{attribute addProperty BoxType "AX8620-0000-0027"}
{attribute addProperty Id "PSM_StatuswordAT %I*PSM_Statusword_C154CB391620WcStateAT %I*WcState_F855686C1620InfoDataAT %I*InfoData_0BDED7BF144180"}
{attribute addProperty CRC "1422836300"}
{attribute addProperty SizeInBites "176"}
{attribute addProperty SizeInBytes "22"}
TYPE AX8620_5E25E4A1 :
STRUCT
	{attribute addProperty Name "PSM_Statusword"}
	PSM_Statusword : PSM_Statusword_C154CB39;
	{attribute addProperty Name "WcState"}
	WcState : WcState_F855686C;
	{attribute addProperty Name "InfoData"}
	InfoData : InfoData_0BDED7BF;
END_STRUCT
END_TYPE

(* stored: Version 1.2.0.0, ProductVersion 3.1.4024.9
   DUT AX8620_5E25E4A1: Id {59ec622a-3ae5-4b67-96d5-5ae8b2e5ce4b} *)
